// TIA Portal V20 export
FUNCTION "Variable_ID" : Void   // FC20226, LAD
TITLE = Any pointer
{ S7_Optimized_Access := 'FALSE' }
// stored: AutoNumber false, SetENOAutomatically false
   VAR_INPUT
      ReadEnable : Bool;
      SelectionIndex : Int;
      VariableLength : Int;
      DB_Source : DB_ANY;
      SourceSize : Int;
      StartAdressSource : Int;
      DB_Destination : DB_ANY;
      DestinationSize : Int;
      StartAdressDestination : Int;
   END_VAR
   VAR_TEMP
      i_dummy : Int;
      i_DB_Source : Int;
      i_DB_Destination : Int;
      di_AdressSource : DInt;
      di_AdressDestination : DInt;
      pa_Any : Any;
      pa_OUT : Any;
   END_VAR
BEGIN

NETWORK
TITLE = Init. Variables
      L     0;
      T     #i_dummy;
//==>
      OPN   #DB_Source;
      L     DBNO;
      T     #i_DB_Source;

//==> OUT01
      OPN   #DB_Destination;
      L     DBNO;
      T     #i_DB_Destination;


NETWORK
TITLE = Read data
      A     #ReadEnable;
      JC    Y_VI;
      JU    N_VI;
Y_VI: NOP   0;
// STRUCTURE:
// BYTE 0  : 10h       -> S7
// BYTE 1  : 13h       -> String
// BYTE 2-3: Length of data
// BYTE 4-5: DB Number
// BYTE 6  : Area 84h=DB
// BYTE 6-8: Startadress

      L     #SelectionIndex;
      L     1;
      -D;
      L     #SourceSize;
      *D;
      L     #StartAdressSource;
      +D;
      T     #di_AdressSource;

      L     P##pa_Any;
      LAR1;

      L     B#16#10;
      T     LB [AR1, P#0.0];
      L     B#16#2;
      T     LB [AR1, P#1.0];
      L     #VariableLength;
      T     LW [AR1, P#2.0];
      L     #i_DB_Source;
      T     LW [AR1, P#4.0];
      L     #di_AdressSource;
      SLD   3;
      OD    DW#16#84000000;
      T     LD [AR1, P#6.0];
//==>
      L     #SelectionIndex;
      L     1;
      -D;
      L     #DestinationSize;
      *D;
      L     #StartAdressDestination;
      +D;
      T     #di_AdressDestination;

      L     P##pa_OUT;
      LAR2;

      L     B#16#10;
      T     LB [AR2, P#0.0];
      L     B#16#2;
      T     LB [AR2, P#1.0];
      L     #VariableLength;
      T     LW [AR2, P#2.0];
      L     #i_DB_Destination;
      T     LW [AR2, P#4.0];
      L     #di_AdressDestination;
      SLD   3;
      OD    DW#16#84000000;
      T     LD [AR2, P#6.0];

//==>Copty to . . .
      CALL  BLKMOV
      ( SRCBLK  := #pa_Any,
        RET_VAL := #i_dummy,
        DSTBLK  := #pa_OUT
      );

N_VI: NOP   0;
END_FUNCTION
